// TIA Portal V21 export
DATA_BLOCK "BatchSAD"   // DB301
{ S7_Optimized_Access := 'FALSE' }
// stored: AutoNumber false
   VAR RETAIN
      BatchStart : Bool;
      BatchEnd : Bool;
      BatchStartPopup : Bool;
      BatchStartPopupYes : Bool;
      BatchStartPopupNo : Bool;
      BatchEndPopup : Bool;
      BatchEndPopupYes : Bool;
      BatchEndPopupNo : Bool;
      Fault : Bool;
      RmAddVesselSafetyPressurePopup : Bool;
      BatchEventString : String;
      BatchStartPopup2 : Bool;
      BatchStartPopup2Ack : Bool;
      ProdTransferFilterSel : Int;   // 0 - FILTER BYPASS 1- THROUGH PF01 2- THROUGH PF02
   END_VAR
BEGIN
END_DATA_BLOCK
